INTERFACE ICUBase

PROPERTY AutomatTask : REFERENCE TO CUBaseAutomat
GET
END_GET
END_PROPERTY

PROPERTY GroundTask : REFERENCE TO CUBaseGround
GET
END_GET
END_PROPERTY

PROPERTY ProcessDataManager : REFERENCE TO ProcessDataManager
GET
END_GET
END_PROPERTY

END_INTERFACE

(* stored: Version 1.1.0.1
   Itf ICUBase: Id {e0435234-64f6-47a6-80fd-c2b672a20857}
   Property AutomatTask: Id {0973134a-28ab-409f-89d6-09a89d3c2b07}
   Get Get: Id {875b00fc-90da-4e77-90bf-2b8bbd7567de}
   Property GroundTask: Id {1d3de518-7983-4b14-bc52-cecc3a9f28ce}
   Get Get: Id {aeb7dbf2-8845-4132-943f-b1517c4d10de}
   Property ProcessDataManager: Id {a36eb78f-c57b-4cc6-9daa-ad73e6b1ba37}
   Get Get: Id {7ae5dbe0-0c01-41d7-9272-ab0df9e64885} *)
